// TIA Portal project "Project1" (V16)

(* hardware
DEVICE "S7-1200 station_1"  S7-1200 Station
   slot 0: "Rack_0"  S7-1200 Rack  Rack  V1.0
   slot 1: "PLC_1"  CPU 1212C AC/DC/Rly  6ES7 212-1BE40-0XB0  V4.4
*)

// ===== PLC "PLC_1"  CPU 1212C AC/DC/Rly =====

VAR_GLOBAL   // PLC tag table "Default tag table"
   "START" AT %I0.1 : Bool;
   "STOP" AT %I0.2 : Bool;
   "MOTOR1" AT %Q0.0 : Bool;
   "MOTOR2" AT %Q0.1 : Bool;
   "TM1" AT %M0.0 : Bool;
   "TM2" AT %M0.1 : Bool;
   "Tag_1" AT %M0.3 : Bool;
   "Tag_2" AT %M0.2 : Bool;
   "Tag_3" AT %M0.5 : Bool;
   "Tag_4" AT %M0.7 : Bool;
   "Tag_5" AT %M0.6 : Bool;
   "Tag_6" AT %M1.2 : Bool;
END_VAR

// folder: System blocks/Program resources

DATA_BLOCK "TIMER1"   // DB1
{ S7_Optimized_Access := 'TRUE' }
AUTHOR : Simatic
FAMILY : IEC
NAME : IEC_TMR
VERSION : 1.0
// stored: InstanceOfName IEC_TIMER
"IEC_TIMER"
BEGIN
END_DATA_BLOCK

DATA_BLOCK "TIMER2"   // DB3
{ S7_Optimized_Access := 'TRUE' }
AUTHOR : Simatic
FAMILY : IEC
NAME : IEC_TMR
VERSION : 1.0
// stored: InstanceOfName IEC_TIMER
"IEC_TIMER"
BEGIN
END_DATA_BLOCK

// folder: (top level)

ORGANIZATION_BLOCK "Main"   // OB1, LAD, ProgramCycle
TITLE = "Main Program Sweep (Cycle)"
{ S7_Optimized_Access := 'TRUE' }
VERSION : 0.1
   VAR_INPUT
      Initial_Call : Bool;   // Initial call of this OB
      Remanence : Bool;   // =True, if remanent data are available
   END_VAR
   VAR_TEMP   // added for the SCL form of the ladder/FBD networks
      _w1 : Bool;
   END_VAR
BEGIN

REGION Network 1
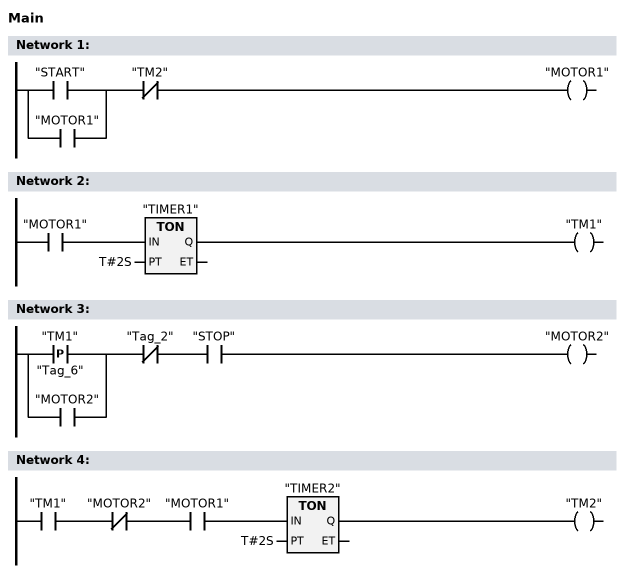
   RUNG wire#powerrail
      Contact( "START" )
      wire#w1
      I_Contact( "TM2" )
      Coil( "MOTOR1" )
   END_RUNG
   RUNG wire#powerrail
      Contact( "MOTOR1" )
   END_RUNG wire#w1
   // the same network as SCL:
   "MOTOR1" := ("START" OR "MOTOR1") AND NOT "TM2";
END_REGION

REGION Network 2
   "TIMER1".TON(IN := "MOTOR1", PT := T#2S);
   "TM1" := "TIMER1".Q;
END_REGION

REGION Network 3
   RUNG wire#powerrail
      P_Contact(operand := "TM1", bit := "Tag_6")
      wire#w1
      I_Contact( "Tag_2" )
      Contact( "STOP" )
      Coil( "MOTOR2" )
   END_RUNG
   RUNG wire#powerrail
      Contact( "MOTOR2" )
   END_RUNG wire#w1
   // the same network as SCL:
   #_w1 := "TM1" AND NOT "Tag_6";   // rising edge of "TM1"
   "Tag_6" := "TM1";
   "MOTOR2" := (#_w1 OR "MOTOR2") AND NOT "Tag_2" AND "STOP";
END_REGION

REGION Network 4
   "TIMER2".TON(IN := "TM1" AND NOT "MOTOR2" AND "MOTOR1", PT := T#2S);
   "TM2" := "TIMER2".Q;
END_REGION
END_ORGANIZATION_BLOCK